// TwinCAT 3 PLC project HFM
// ProgramVersion: 3.1.4024.0
// libraries:
//   Tc2_Standard, * (Beckhoff Automation GmbH)
//   Tc2_System, * (Beckhoff Automation GmbH)
//   Tc3_Module, * (Beckhoff Automation GmbH)
//   LCLS General,0.0.0,SLAC
//   lcls-twincat-motion,0.0.0,SLAC
//   PMPS,0.0.0,SLAC - LCLS
//   TcUnit,1.3.0.0,www.tcunit.org
// project tree:
//   / PlcTask.TcTTO
//   POUs/ MAIN.TcPOU
// real-time tasks:
//   TASK PlcTask: cycle T#10ms, priority 20, ADS port 350
// motion (NC):
//   TASK NC-Task 1 SAF: cycle T#2ms, priority 4, ADS port 501
//   TASK NC-Task 1 SVB: cycle T#10ms, priority 8, ADS port 511
//   AXIS Axis 1(HFM-Y1) (id 1)
//     Dynamic: AccelerationMaximum=20, DecelerationMaximum=20, Acceleration=0.742063, Deceleration=0.742063, Jerk=275.329
//     Velo: RefSearch=5, RefSync=5, SlowManual=5, FastManual=5, Maximum=0.2
//     PositionAreaControl: Range=0.0002
//     MotionControl: Range=0.5, Time=1
//     TargetPosControl: Range=0.0001
//     PEHControl: Time=0.1
//     OtherSettings: AllowMotionCmdToSlave=true, PulseDistancePos=0.5, PulseDistanceNeg=0.5
//     encoder EncType=4
//       EncPara: ScaleFactorNumerator=0.0002, Inverse=true, MaxCount=#xffffffff
//     drive DrvType=5
//       DrvPara: Inverse=true
//         Analog: VeloReferenz=20, TorqueSetpointScale=10, ScaleFactorActTorque=0.1
//         TimeComp: TaskDelayCycles=1
//     controller CtrType=1
//       CtrPara: PriorControlFactor=1
//         PosDiffControl: Range=1
//         PID: PosKp=22
//         Observer: BandWidth=20
//   AXIS Axis 2(HFM-Y2) (id 2)
//     Dynamic: AccelerationMaximum=20, DecelerationMaximum=20, Acceleration=0.75757, Deceleration=0.75757, Jerk=286.956
//     Velo: RefSearch=5, RefSync=5, SlowManual=5, FastManual=5, Maximum=0.2
//     PositionAreaControl: Range=0.0002
//     TargetPosControl: Range=0.0001
//     OtherSettings: AllowMotionCmdToSlave=true, PulseDistancePos=0.5, PulseDistanceNeg=0.5
//     encoder EncType=4
//       EncPara: ScaleFactorNumerator=0.0002, Inverse=true, MaxCount=#xffffffff
//     drive DrvType=5
//       DrvPara: Inverse=true
//         Analog: VeloReferenz=20, TorqueSetpointScale=10, ScaleFactorActTorque=0.1
//         TimeComp: TaskDelayCycles=1
//     controller CtrType=1
//       CtrPara: PriorControlFactor=1
//         PosDiffControl: Range=2
//         PID: PosKp=22
//         Observer: BandWidth=20
//   AXIS Axis 3(HFM-Y3) (id 3)
//     Dynamic: AccelerationMaximum=20, DecelerationMaximum=20, Acceleration=0.742063, Deceleration=0.742063, Jerk=275.329
//     Velo: RefSearch=5, RefSync=5, SlowManual=5, FastManual=5, Maximum=0.2
//     PositionAreaControl: Range=0.0002
//     TargetPosControl: Range=0.0001
//     OtherSettings: AllowMotionCmdToSlave=true, PulseDistancePos=0.5, PulseDistanceNeg=0.5
//     encoder EncType=4
//       EncPara: ScaleFactorNumerator=0.0002, Inverse=true, MaxCount=#xffffffff
//     drive DrvType=5
//       DrvPara: Inverse=true
//         Analog: VeloReferenz=20, TorqueSetpointScale=10, ScaleFactorActTorque=0.1
//         TimeComp: TaskDelayCycles=1
//     controller CtrType=1
//       CtrPara: PriorControlFactor=1
//         PosDiffControl: Range=2
//         PID: PosKp=22
//         Observer: BandWidth=20
//   AXIS Axis 4(HFM-X1) (id 4)
//     Dynamic: AccelerationMaximum=20, DecelerationMaximum=20, Acceleration=6.71181, Deceleration=6.71181, Jerk=22524.2
//     Velo: RefSearch=5, RefSync=5, SlowManual=5, FastManual=5, Maximum=0.2
//     PositionAreaControl: Range=2e-05
//     TargetPosControl: Range=1e-05
//     OtherSettings: AllowMotionCmdToSlave=true, PulseDistancePos=0.5, PulseDistanceNeg=0.5
//     encoder EncType=4
//       EncPara: ScaleFactorNumerator=2e-05, MaxCount=#xffffffff
//     drive DrvType=5
//       Analog: VeloReferenz=20, TorqueSetpointScale=10, ScaleFactorActTorque=0.1
//       TimeComp: TaskDelayCycles=1
//     controller CtrType=1
//       CtrPara: PriorControlFactor=1
//         PID: PosKp=50
//         Observer: BandWidth=20
//   AXIS Axis 5(HFM-X2) (id 5)
//     Dynamic: AccelerationMaximum=20, DecelerationMaximum=20, Acceleration=3.45558, Deceleration=3.45558, Jerk=5970.51
//     Velo: RefSearch=5, RefSync=5, SlowManual=5, FastManual=5, Maximum=0.2
//     PositionAreaControl: Range=2e-05
//     TargetPosControl: Range=1e-05
//     OtherSettings: AllowMotionCmdToSlave=true, PulseDistancePos=0.5, PulseDistanceNeg=0.5
//     encoder EncType=4
//       EncPara: ScaleFactorNumerator=2e-05, MaxCount=#xffffffff
//     drive DrvType=5
//       Analog: VeloReferenz=20, TorqueSetpointScale=10, ScaleFactorActTorque=0.1
//       TimeComp: TaskDelayCycles=1
//     controller CtrType=1
//       CtrPara: PriorControlFactor=1
//         PID: PosKp=50
//         Observer: BandWidth=20
//   AXIS Axis 6(FM-Y1) (id 6)
//     Dynamic: AccelerationMaximum=20, DecelerationMaximum=20, Acceleration=0.742063, Deceleration=0.742063, Jerk=275.329
//     Velo: RefSearch=1, RefSync=1, SlowManual=1, FastManual=1, Maximum=0.2
//     PositionAreaControl: Range=0.0002
//     TargetPosControl: Range=0.0001
//     OtherSettings: AllowMotionCmdToSlave=true, PulseDistancePos=0.5, PulseDistanceNeg=0.5
//     encoder EncType=4
//       EncPara: ScaleFactorNumerator=0.0002, Inverse=true, MaxCount=#xffffffff
//     drive DrvType=5
//       DrvPara: Inverse=true
//         Analog: VeloReferenz=20, TorqueSetpointScale=10, ScaleFactorActTorque=0.1
//         TimeComp: TaskDelayCycles=1
//     controller CtrType=1
//       CtrPara: PriorControlFactor=1
//         PosDiffControl: Range=1
//         PID: PosKp=22
//         Observer: BandWidth=20
//   AXIS Axis 7(FM-Y2) (id 7)
//     Dynamic: AccelerationMaximum=20, DecelerationMaximum=20, Acceleration=0.742063, Deceleration=0.742063, Jerk=275.329
//     Velo: RefSearch=1, RefSync=1, SlowManual=1, FastManual=1, Maximum=0.2
//     PositionAreaControl: Range=0.0002
//     TargetPosControl: Range=0.0001
//     OtherSettings: AllowMotionCmdToSlave=true, PulseDistancePos=0.5, PulseDistanceNeg=0.5
//     encoder EncType=4
//       EncPara: ScaleFactorNumerator=0.0002, Inverse=true, MaxCount=#xffffffff
//     drive DrvType=5
//       DrvPara: Inverse=true
//         Analog: VeloReferenz=20, TorqueSetpointScale=10, ScaleFactorActTorque=0.1
//         TimeComp: TaskDelayCycles=1
//     controller CtrType=1
//       CtrPara: PriorControlFactor=1
//         PosDiffControl: Range=1
//         PID: PosKp=22
//         Observer: BandWidth=20
//   AXIS Axis 8(FM-Y3) (id 8)
//     Dynamic: AccelerationMaximum=20, DecelerationMaximum=20, Acceleration=0.742063, Deceleration=0.742063, Jerk=275.329
//     Velo: RefSearch=1, RefSync=1, SlowManual=1, FastManual=1, Maximum=0.2
//     PositionAreaControl: Range=0.0002
//     TargetPosControl: Range=0.0001
//     OtherSettings: AllowMotionCmdToSlave=true, PulseDistancePos=0.5, PulseDistanceNeg=0.5
//     encoder EncType=4
//       EncPara: ScaleFactorNumerator=0.0002, Inverse=true, MaxCount=#xffffffff
//     drive DrvType=5
//       DrvPara: Inverse=true
//         Analog: VeloReferenz=20, TorqueSetpointScale=10, ScaleFactorActTorque=0.1
//         TimeComp: TaskDelayCycles=1
//     controller CtrType=1
//       CtrPara: PriorControlFactor=1
//         PosDiffControl: Range=1
//         PID: PosKp=22
//         Observer: BandWidth=20
//   AXIS Axis 9(FM-X1) (id 9)
//     Dynamic: AccelerationMaximum=20, DecelerationMaximum=20, Acceleration=6.71181, Deceleration=6.71181, Jerk=22524.2
//     Velo: RefSearch=1, RefSync=1, SlowManual=1, FastManual=1, Maximum=0.2
//     PositionAreaControl: Range=2e-05
//     TargetPosControl: Range=1e-05
//     OtherSettings: AllowMotionCmdToSlave=true, PulseDistancePos=0.5, PulseDistanceNeg=0.5
//     encoder EncType=4
//       EncPara: ScaleFactorNumerator=2e-05, MaxCount=#xffffffff
//     drive DrvType=5
//       Analog: VeloReferenz=20, TorqueSetpointScale=10, ScaleFactorActTorque=0.1
//       TimeComp: TaskDelayCycles=1
//     controller CtrType=1
//       CtrPara: PriorControlFactor=1
//         PID: PosKp=50
//         Observer: BandWidth=20
//   AXIS Axis 10(FM-X2) (id 10)
//     Dynamic: AccelerationMaximum=20, DecelerationMaximum=20, Acceleration=6.71181, Deceleration=6.71181, Jerk=22524.2
//     Velo: RefSearch=1, RefSync=1, SlowManual=1, FastManual=1, Maximum=0.2
//     PositionAreaControl: Range=2e-05
//     TargetPosControl: Range=1e-05
//     OtherSettings: AllowMotionCmdToSlave=true, PulseDistancePos=0.5, PulseDistanceNeg=0.5
//     encoder EncType=4
//       EncPara: ScaleFactorNumerator=2e-05, MaxCount=#xffffffff
//     drive DrvType=5
//       Analog: VeloReferenz=20, TorqueSetpointScale=10, ScaleFactorActTorque=0.1
//       TimeComp: TaskDelayCycles=1
//     controller CtrType=1
//       CtrPara: PriorControlFactor=1
//         PID: PosKp=50
//         Observer: BandWidth=20
// I/O:
//   DEVICE Device 3 (EtherCAT), AmsNetId 169.254.61.1.4.1
//     Term 1 (EK1100) [EK1100 EtherCAT Coupler (2A E-Bus)]
//       Term 2 (EL2522) [EL2522 2Ch. Pulse Train Output]
//       Term 3 (EL5112) [EL5112 2Ch. Inc. Encoder 5V (2xAB or 1xABC RS422,TTL)]
//       Term 4 (EL2522) [EL2522 2Ch. Pulse Train Output]
//       Term 5 (EL5112) [EL5112 2Ch. Inc. Encoder 5V (2xAB or 1xABC RS422,TTL)]
//       Term 6 (EL2522) [EL2522 2Ch. Pulse Train Output]
//       Term 7 (EL1889) [EL1889 16Ch. Dig. Input 24V, 3ms, negative]
//       Term 8 (EL9011) [EL9011 End Terminal]
//   DEVICE Device 1 (EtherCAT), AmsNetId 192.168.61.50.2.1
//     Term 9 (EK1100) [EK1100 EtherCAT Coupler (2A E-Bus)]
//       Term 10 (EL2522) [EL2522 2Ch. Pulse Train Output]
//       Term 11 (EL5112) [EL5112 2Ch. Inc. Encoder 5V (2xAB or 1xABC RS422,TTL)]
//       Term 12 (EL2522) [EL2522 2Ch. Pulse Train Output]
//       Term 13 (EL5112) [EL5112 2Ch. Inc. Encoder 5V (2xAB or 1xABC RS422,TTL)]
//       Term 14 (EL2522) [EL2522 2Ch. Pulse Train Output]
//       Term 15 (EL1889) [EL1889 16Ch. Dig. Input 24V, 3ms, negative]
//       Term 8 (EL9011) [EL9011 End Terminal]
// variable links:
//   NC-Task 1 SAF/Axes/Axis 10(FM-X2) <-> Device 1 (EtherCAT)/Term 9 (EK1100)/Term 14 (EL2522)
//     Drive/Inputs/In/nState1 @bit 6 <-> PTO Status Channel 1/Status/Error
//     Drive/Inputs/In/nState1 @bit 1 <-> PTO Status Channel 1/Status/Ramp active
//     Drive/Inputs/In/nState1 <-> PTO Status Channel 1/Status/Sel. Ack/End counter
//     Drive/Inputs/In/nState2 @bit 5 <-> PTO Status Channel 1/Status/Sync error
//     Drive/Inputs/In/nState2 @bit 7 <-> PTO Status Channel 1/Status/TxPDO Toggle
//     Drive/Inputs/In/nState4 @bit 1 <-> WcState/InputToggle
//     Drive/Inputs/In/nState4 <-> WcState/WcState
//     Drive/Outputs/Out/nCtrl1 @bit 1 <-> PTO Control Channel 1/Control/Disable ramp
//     Drive/Outputs/Out/nCtrl1 <-> PTO Control Channel 1/Control/Frequency select
//     Drive/Outputs/Out/nCtrl1 @bit 2 <-> PTO Control Channel 1/Control/Go counter
//     Drive/Outputs/Out/nDataOut1[0] <-> PTO Control Channel 1/Frequency value
//     Drive/Outputs/Out/nDataOut5 <-> PTO Target Channel 1/Target counter value
//     Enc/Inputs/In/nDataIn1 <-> ENC Status Channel 1/Counter value
//     Enc/Inputs/In/nState1 @bit 4 <-> ENC Status Channel 1/Status/Counter overflow
//     Enc/Inputs/In/nState1 @bit 3 <-> ENC Status Channel 1/Status/Counter underflow
//     Enc/Inputs/In/nState1 @bit 2 <-> ENC Status Channel 1/Status/Set counter done
//     Enc/Inputs/In/nState2 @bit 5 <-> ENC Status Channel 1/Status/Sync error
//     Enc/Inputs/In/nState2 @bit 6 <-> ENC Status Channel 1/Status/TxPDO State
//     Enc/Inputs/In/nState2 @bit 7 <-> ENC Status Channel 1/Status/TxPDO Toggle
//     Enc/Inputs/In/nState4 @bit 1 <-> WcState/InputToggle
//     Enc/Inputs/In/nState4 <-> WcState/WcState
//     Enc/Outputs/Out/nCtrl1 @bit 2 <-> ENC Control Channel 1/Control/Set counter
//     Enc/Outputs/Out/nCtrl2 @bit 7 <-> ENC Control Channel 1/Control/Reserved
//     Enc/Outputs/Out/nDataOut1 <-> ENC Control Channel 1/Set counter value
//   NC-Task 1 SAF/Axes/Axis 2(HFM-Y2) <-> Device 3 (EtherCAT)/Term 1 (EK1100)/Term 2 (EL2522)
//     Drive/Inputs/In/nState1 @bit 6 <-> PTO Status Channel 2/Status/Error
//     Drive/Inputs/In/nState1 @bit 1 <-> PTO Status Channel 2/Status/Ramp active
//     Drive/Inputs/In/nState1 <-> PTO Status Channel 2/Status/Sel. Ack/End counter
//     Drive/Inputs/In/nState2 @bit 5 <-> PTO Status Channel 2/Status/Sync error
//     Drive/Inputs/In/nState2 @bit 7 <-> PTO Status Channel 2/Status/TxPDO Toggle
//     Drive/Inputs/In/nState4 @bit 1 <-> WcState/InputToggle
//     Drive/Inputs/In/nState4 <-> WcState/WcState
//     Drive/Outputs/Out/nCtrl1 @bit 1 <-> PTO Control Channel 2/Control/Disable ramp
//     Drive/Outputs/Out/nCtrl1 <-> PTO Control Channel 2/Control/Frequency select
//     Drive/Outputs/Out/nCtrl1 @bit 2 <-> PTO Control Channel 2/Control/Go counter
//     Drive/Outputs/Out/nDataOut1[0] <-> PTO Control Channel 2/Frequency value
//     Drive/Outputs/Out/nDataOut5 <-> PTO Target Channel 2/Target counter value
//   NC-Task 1 SAF/Axes/Axis 2(HFM-Y2) <-> Device 3 (EtherCAT)/Term 1 (EK1100)/Term 3 (EL5112)
//     Enc/Inputs/In/nDataIn1 <-> ENC Status Channel 2/Counter value
//     Enc/Inputs/In/nDataIn2 <-> ENC Status Channel 2/Latch value
//     Enc/Inputs/In/nState1 @bit 4 <-> ENC Status Channel 2/Status/Counter overflow
//     Enc/Inputs/In/nState1 @bit 3 <-> ENC Status Channel 2/Status/Counter underflow
//     Enc/Inputs/In/nState1 @bit 1 <-> ENC Status Channel 2/Status/Latch extern valid
//     Enc/Inputs/In/nState1 @bit 6 <-> ENC Status Channel 2/Status/Open circuit
//     Enc/Inputs/In/nState1 @bit 2 <-> ENC Status Channel 2/Status/Set counter done
//     Enc/Inputs/In/nState2 @bit 4 <-> ENC Status Channel 2/Status/Diag
//     Enc/Inputs/In/nState2 @bit 6 <-> ENC Status Channel 2/Status/Input cycle counter
//     Enc/Inputs/In/nState2 <-> ENC Status Channel 2/Status/Status of input A
//     Enc/Inputs/In/nState2 @bit 1 <-> ENC Status Channel 2/Status/Status of input B
//     Enc/Inputs/In/nState2 @bit 3 <-> ENC Status Channel 2/Status/Status of input gate
//     Enc/Inputs/In/nState2 @bit 5 <-> ENC Status Channel 2/Status/TxPDO State
//     Enc/Inputs/In/nState3 @bit 4 <-> ENC Status Channel 2/Status/Counter value out of range
//     Enc/Inputs/In/nState3 <-> ENC Status Channel 2/Status/Software gate valid
//     Enc/Inputs/In/nState4 @bit 1 <-> WcState/InputToggle
//     Enc/Inputs/In/nState4 <-> WcState/WcState
//     Enc/Outputs/Out/nCtrl1 @bit 3 <-> ENC Control Channel 2/Control/Enable latch extern on negative edge
//     Enc/Outputs/Out/nCtrl1 @bit 1 <-> ENC Control Channel 2/Control/Enable latch extern on positive edge
//     Enc/Outputs/Out/nCtrl1 @bit 2 <-> ENC Control Channel 2/Control/Set counter
//     Enc/Outputs/Out/nCtrl2 @bit 2 <-> ENC Control Channel 2/Control/Set counter on latch extern on negative edge
//     Enc/Outputs/Out/nCtrl2 @bit 1 <-> ENC Control Channel 2/Control/Set counter on latch extern on positive edge
//     Enc/Outputs/Out/nCtrl2 <-> ENC Control Channel 2/Control/Set software gate
//     Enc/Outputs/Out/nDataOut1 <-> ENC Control Channel 2/Set counter value
//   NC-Task 1 SAF/Axes/Axis 3(HFM-Y3) <-> Device 3 (EtherCAT)/Term 1 (EK1100)/Term 4 (EL2522)
//     Drive/Inputs/In/nState1 @bit 6 <-> PTO Status Channel 1/Status/Error
//     Drive/Inputs/In/nState1 @bit 1 <-> PTO Status Channel 1/Status/Ramp active
//     Drive/Inputs/In/nState1 <-> PTO Status Channel 1/Status/Sel. Ack/End counter
//     Drive/Inputs/In/nState2 @bit 5 <-> PTO Status Channel 1/Status/Sync error
//     Drive/Inputs/In/nState2 @bit 7 <-> PTO Status Channel 1/Status/TxPDO Toggle
//     Drive/Inputs/In/nState4 @bit 1 <-> WcState/InputToggle
//     Drive/Inputs/In/nState4 <-> WcState/WcState
//     Drive/Outputs/Out/nCtrl1 @bit 1 <-> PTO Control Channel 1/Control/Disable ramp
//     Drive/Outputs/Out/nCtrl1 <-> PTO Control Channel 1/Control/Frequency select
//     Drive/Outputs/Out/nCtrl1 @bit 2 <-> PTO Control Channel 1/Control/Go counter
//     Drive/Outputs/Out/nDataOut1[0] <-> PTO Control Channel 1/Frequency value
//     Drive/Outputs/Out/nDataOut5 <-> PTO Target Channel 1/Target counter value
//   NC-Task 1 SAF/Axes/Axis 3(HFM-Y3) <-> Device 3 (EtherCAT)/Term 1 (EK1100)/Term 5 (EL5112)
//     Enc/Inputs/In/nDataIn1 <-> ENC Status Channel 1/Counter value
//     Enc/Inputs/In/nDataIn2 <-> ENC Status Channel 1/Latch value
//     Enc/Inputs/In/nState1 @bit 4 <-> ENC Status Channel 1/Status/Counter overflow
//     Enc/Inputs/In/nState1 @bit 3 <-> ENC Status Channel 1/Status/Counter underflow
//     Enc/Inputs/In/nState1 @bit 7 <-> ENC Status Channel 1/Status/Extrapolation stall
//     Enc/Inputs/In/nState1 <-> ENC Status Channel 1/Status/Latch C valid
//     Enc/Inputs/In/nState1 @bit 1 <-> ENC Status Channel 1/Status/Latch extern valid
//     Enc/Inputs/In/nState1 @bit 6 <-> ENC Status Channel 1/Status/Open circuit
//     Enc/Inputs/In/nState1 @bit 2 <-> ENC Status Channel 1/Status/Set counter done
//     Enc/Inputs/In/nState1 @bit 5 <-> ENC Status Channel 1/Status/Status of input status
//     Enc/Inputs/In/nState2 @bit 4 <-> ENC Status Channel 1/Status/Diag
//     Enc/Inputs/In/nState2 @bit 6 <-> ENC Status Channel 1/Status/Input cycle counter
//     Enc/Inputs/In/nState2 <-> ENC Status Channel 1/Status/Status of input A
//     Enc/Inputs/In/nState2 @bit 1 <-> ENC Status Channel 1/Status/Status of input B
//     Enc/Inputs/In/nState2 @bit 2 <-> ENC Status Channel 1/Status/Status of input C
//     Enc/Inputs/In/nState2 @bit 3 <-> ENC Status Channel 1/Status/Status of input gate
//     Enc/Inputs/In/nState2 @bit 5 <-> ENC Status Channel 1/Status/TxPDO State
//     Enc/Inputs/In/nState3 @bit 4 <-> ENC Status Channel 1/Status/Counter value out of range
//     Enc/Inputs/In/nState3 @bit 2 <-> ENC Status Channel 1/Status/Direction inversion detected
//     Enc/Inputs/In/nState3 @bit 1 <-> ENC Status Channel 1/Status/Latch extern 2 valid
//     Enc/Inputs/In/nState3 <-> ENC Status Channel 1/Status/Software gate valid
//     Enc/Inputs/In/nState3 @bit 3 <-> ENC Status Channel 1/Status/Status of extern latch
//     Enc/Inputs/In/nState4 @bit 1 <-> WcState/InputToggle
//     Enc/Inputs/In/nState4 <-> WcState/WcState
//     Enc/Outputs/Out/nCtrl1 <-> ENC Control Channel 1/Control/Enable latch C
//     Enc/Outputs/Out/nCtrl1 @bit 3 <-> ENC Control Channel 1/Control/Enable latch extern on negative edge
//     Enc/Outputs/Out/nCtrl1 @bit 1 <-> ENC Control Channel 1/Control/Enable latch extern on positive edge
//     Enc/Outputs/Out/nCtrl1 @bit 2 <-> ENC Control Channel 1/Control/Set counter
//     Enc/Outputs/Out/nCtrl1 @bit 7 <-> ENC Control Channel 1/Control/Set counter on latch C
//     Enc/Outputs/Out/nCtrl2 @bit 4 <-> ENC Control Channel 1/Control/Enable latch extern 2 on negative edge
//     Enc/Outputs/Out/nCtrl2 @bit 3 <-> ENC Control Channel 1/Control/Enable latch extern 2 on positive edge
//     Enc/Outputs/Out/nCtrl2 @bit 2 <-> ENC Control Channel 1/Control/Set counter on latch extern on negative edge
//     Enc/Outputs/Out/nCtrl2 @bit 1 <-> ENC Control Channel 1/Control/Set counter on latch extern on positive edge
//     Enc/Outputs/Out/nCtrl2 <-> ENC Control Channel 1/Control/Set software gate
//     Enc/Outputs/Out/nDataOut1 <-> ENC Control Channel 1/Set counter value
//   NC-Task 1 SAF/Axes/Axis 4(HFM-X1) <-> Device 3 (EtherCAT)/Term 1 (EK1100)/Term 4 (EL2522)
//     Drive/Inputs/In/nState1 @bit 6 <-> PTO Status Channel 2/Status/Error
//     Drive/Inputs/In/nState1 @bit 1 <-> PTO Status Channel 2/Status/Ramp active
//     Drive/Inputs/In/nState1 <-> PTO Status Channel 2/Status/Sel. Ack/End counter
//     Drive/Inputs/In/nState2 @bit 5 <-> PTO Status Channel 2/Status/Sync error
//     Drive/Inputs/In/nState2 @bit 7 <-> PTO Status Channel 2/Status/TxPDO Toggle
//     Drive/Inputs/In/nState4 @bit 1 <-> WcState/InputToggle
//     Drive/Inputs/In/nState4 <-> WcState/WcState
//     Drive/Outputs/Out/nCtrl1 @bit 1 <-> PTO Control Channel 2/Control/Disable ramp
//     Drive/Outputs/Out/nCtrl1 <-> PTO Control Channel 2/Control/Frequency select
//     Drive/Outputs/Out/nCtrl1 @bit 2 <-> PTO Control Channel 2/Control/Go counter
//     Drive/Outputs/Out/nDataOut1[0] <-> PTO Control Channel 2/Frequency value
//     Drive/Outputs/Out/nDataOut5 <-> PTO Target Channel 2/Target counter value
//     Enc/Inputs/In/nDataIn1 <-> ENC Status Channel 2/Counter value
//     Enc/Inputs/In/nState1 @bit 4 <-> ENC Status Channel 2/Status/Counter overflow
//     Enc/Inputs/In/nState1 @bit 3 <-> ENC Status Channel 2/Status/Counter underflow
//     Enc/Inputs/In/nState1 @bit 2 <-> ENC Status Channel 2/Status/Set counter done
//     Enc/Inputs/In/nState2 @bit 5 <-> ENC Status Channel 2/Status/Sync error
//     Enc/Inputs/In/nState2 @bit 6 <-> ENC Status Channel 2/Status/TxPDO State
//     Enc/Inputs/In/nState2 @bit 7 <-> ENC Status Channel 2/Status/TxPDO Toggle
//     Enc/Inputs/In/nState4 @bit 1 <-> WcState/InputToggle
//     Enc/Inputs/In/nState4 <-> WcState/WcState
//     Enc/Outputs/Out/nCtrl1 @bit 2 <-> ENC Control Channel 2/Control/Set counter
//     Enc/Outputs/Out/nCtrl2 @bit 7 <-> ENC Control Channel 2/Control/Reserved
//     Enc/Outputs/Out/nDataOut1 <-> ENC Control Channel 2/Set counter value
//   NC-Task 1 SAF/Axes/Axis 5(HFM-X2) <-> Device 3 (EtherCAT)/Term 1 (EK1100)/Term 6 (EL2522)
//     Drive/Inputs/In/nState1 @bit 6 <-> PTO Status Channel 1/Status/Error
//     Drive/Inputs/In/nState1 @bit 1 <-> PTO Status Channel 1/Status/Ramp active
//     Drive/Inputs/In/nState1 <-> PTO Status Channel 1/Status/Sel. Ack/End counter
//     Drive/Inputs/In/nState2 @bit 5 <-> PTO Status Channel 1/Status/Sync error
//     Drive/Inputs/In/nState2 @bit 7 <-> PTO Status Channel 1/Status/TxPDO Toggle
//     Drive/Inputs/In/nState4 @bit 1 <-> WcState/InputToggle
//     Drive/Inputs/In/nState4 <-> WcState/WcState
//     Drive/Outputs/Out/nCtrl1 @bit 1 <-> PTO Control Channel 1/Control/Disable ramp
//     Drive/Outputs/Out/nCtrl1 <-> PTO Control Channel 1/Control/Frequency select
//     Drive/Outputs/Out/nCtrl1 @bit 2 <-> PTO Control Channel 1/Control/Go counter
//     Drive/Outputs/Out/nDataOut1[0] <-> PTO Control Channel 1/Frequency value
//     Drive/Outputs/Out/nDataOut5 <-> PTO Target Channel 1/Target counter value
//     Enc/Inputs/In/nDataIn1 <-> ENC Status Channel 1/Counter value
//     Enc/Inputs/In/nState1 @bit 4 <-> ENC Status Channel 1/Status/Counter overflow
//     Enc/Inputs/In/nState1 @bit 3 <-> ENC Status Channel 1/Status/Counter underflow
//     Enc/Inputs/In/nState1 @bit 2 <-> ENC Status Channel 1/Status/Set counter done
//     Enc/Inputs/In/nState2 @bit 5 <-> ENC Status Channel 1/Status/Sync error
//     Enc/Inputs/In/nState2 @bit 6 <-> ENC Status Channel 1/Status/TxPDO State
//     Enc/Inputs/In/nState2 @bit 7 <-> ENC Status Channel 1/Status/TxPDO Toggle
//     Enc/Inputs/In/nState4 @bit 1 <-> WcState/InputToggle
//     Enc/Inputs/In/nState4 <-> WcState/WcState
//     Enc/Outputs/Out/nCtrl1 @bit 2 <-> ENC Control Channel 1/Control/Set counter
//     Enc/Outputs/Out/nCtrl2 @bit 7 <-> ENC Control Channel 1/Control/Reserved
//     Enc/Outputs/Out/nDataOut1 <-> ENC Control Channel 1/Set counter value
//   NC-Task 1 SAF/Axes/Axis 6(FM-Y1) <-> Device 1 (EtherCAT)/Term 9 (EK1100)/Term 10 (EL2522)
//     Drive/Inputs/In/nState1 @bit 6 <-> PTO Status Channel 1/Status/Error
//     Drive/Inputs/In/nState1 @bit 1 <-> PTO Status Channel 1/Status/Ramp active
//     Drive/Inputs/In/nState1 <-> PTO Status Channel 1/Status/Sel. Ack/End counter
//     Drive/Inputs/In/nState2 @bit 5 <-> PTO Status Channel 1/Status/Sync error
//     Drive/Inputs/In/nState2 @bit 7 <-> PTO Status Channel 1/Status/TxPDO Toggle
//     Drive/Inputs/In/nState4 @bit 1 <-> WcState/InputToggle
//     Drive/Inputs/In/nState4 <-> WcState/WcState
//     Drive/Outputs/Out/nCtrl1 @bit 1 <-> PTO Control Channel 1/Control/Disable ramp
//     Drive/Outputs/Out/nCtrl1 <-> PTO Control Channel 1/Control/Frequency select
//     Drive/Outputs/Out/nCtrl1 @bit 2 <-> PTO Control Channel 1/Control/Go counter
//     Drive/Outputs/Out/nDataOut1[0] <-> PTO Control Channel 1/Frequency value
//     Drive/Outputs/Out/nDataOut5 <-> PTO Target Channel 1/Target counter value
//   NC-Task 1 SAF/Axes/Axis 6(FM-Y1) <-> Device 1 (EtherCAT)/Term 9 (EK1100)/Term 11 (EL5112)
//     Enc/Inputs/In/nDataIn1 <-> ENC Status Channel 1/Counter value
//     Enc/Inputs/In/nDataIn2 <-> ENC Status Channel 1/Latch value
//     Enc/Inputs/In/nState1 @bit 4 <-> ENC Status Channel 1/Status/Counter overflow
//     Enc/Inputs/In/nState1 @bit 3 <-> ENC Status Channel 1/Status/Counter underflow
//     Enc/Inputs/In/nState1 @bit 1 <-> ENC Status Channel 1/Status/Latch extern valid
//     Enc/Inputs/In/nState1 @bit 6 <-> ENC Status Channel 1/Status/Open circuit
//     Enc/Inputs/In/nState1 @bit 2 <-> ENC Status Channel 1/Status/Set counter done
//     Enc/Inputs/In/nState2 @bit 4 <-> ENC Status Channel 1/Status/Diag
//     Enc/Inputs/In/nState2 @bit 6 <-> ENC Status Channel 1/Status/Input cycle counter
//     Enc/Inputs/In/nState2 <-> ENC Status Channel 1/Status/Status of input A
//     Enc/Inputs/In/nState2 @bit 1 <-> ENC Status Channel 1/Status/Status of input B
//     Enc/Inputs/In/nState2 @bit 3 <-> ENC Status Channel 1/Status/Status of input gate
//     Enc/Inputs/In/nState2 @bit 5 <-> ENC Status Channel 1/Status/TxPDO State
//     Enc/Inputs/In/nState3 @bit 4 <-> ENC Status Channel 1/Status/Counter value out of range
//     Enc/Inputs/In/nState3 <-> ENC Status Channel 1/Status/Software gate valid
//     Enc/Inputs/In/nState4 @bit 1 <-> WcState/InputToggle
//     Enc/Inputs/In/nState4 <-> WcState/WcState
//     Enc/Outputs/Out/nCtrl1 @bit 3 <-> ENC Control Channel 1/Control/Enable latch extern on negative edge
//     Enc/Outputs/Out/nCtrl1 @bit 1 <-> ENC Control Channel 1/Control/Enable latch extern on positive edge
//     Enc/Outputs/Out/nCtrl1 @bit 2 <-> ENC Control Channel 1/Control/Set counter
//     Enc/Outputs/Out/nCtrl2 @bit 2 <-> ENC Control Channel 1/Control/Set counter on latch extern on negative edge
//     Enc/Outputs/Out/nCtrl2 @bit 1 <-> ENC Control Channel 1/Control/Set counter on latch extern on positive edge
//     Enc/Outputs/Out/nCtrl2 <-> ENC Control Channel 1/Control/Set software gate
//     Enc/Outputs/Out/nDataOut1 <-> ENC Control Channel 1/Set counter value
//   NC-Task 1 SAF/Axes/Axis 7(FM-Y2) <-> Device 1 (EtherCAT)/Term 9 (EK1100)/Term 10 (EL2522)
//     Drive/Inputs/In/nState1 @bit 6 <-> PTO Status Channel 2/Status/Error
//     Drive/Inputs/In/nState1 @bit 1 <-> PTO Status Channel 2/Status/Ramp active
//     Drive/Inputs/In/nState1 <-> PTO Status Channel 2/Status/Sel. Ack/End counter
//     Drive/Inputs/In/nState2 @bit 5 <-> PTO Status Channel 2/Status/Sync error
//     Drive/Inputs/In/nState2 @bit 7 <-> PTO Status Channel 2/Status/TxPDO Toggle
//     Drive/Inputs/In/nState4 @bit 1 <-> WcState/InputToggle
//     Drive/Inputs/In/nState4 <-> WcState/WcState
//     Drive/Outputs/Out/nCtrl1 @bit 1 <-> PTO Control Channel 2/Control/Disable ramp
//     Drive/Outputs/Out/nCtrl1 <-> PTO Control Channel 2/Control/Frequency select
//     Drive/Outputs/Out/nCtrl1 @bit 2 <-> PTO Control Channel 2/Control/Go counter
//     Drive/Outputs/Out/nDataOut1[0] <-> PTO Control Channel 2/Frequency value
//     Drive/Outputs/Out/nDataOut5 <-> PTO Target Channel 2/Target counter value
//   NC-Task 1 SAF/Axes/Axis 7(FM-Y2) <-> Device 1 (EtherCAT)/Term 9 (EK1100)/Term 11 (EL5112)
//     Enc/Inputs/In/nDataIn1 <-> ENC Status Channel 2/Counter value
//     Enc/Inputs/In/nDataIn2 <-> ENC Status Channel 2/Latch value
//     Enc/Inputs/In/nState1 @bit 4 <-> ENC Status Channel 2/Status/Counter overflow
//     Enc/Inputs/In/nState1 @bit 3 <-> ENC Status Channel 2/Status/Counter underflow
//     Enc/Inputs/In/nState1 @bit 1 <-> ENC Status Channel 2/Status/Latch extern valid
//     Enc/Inputs/In/nState1 @bit 6 <-> ENC Status Channel 2/Status/Open circuit
//     Enc/Inputs/In/nState1 @bit 2 <-> ENC Status Channel 2/Status/Set counter done
//     Enc/Inputs/In/nState2 @bit 4 <-> ENC Status Channel 2/Status/Diag
//     Enc/Inputs/In/nState2 @bit 6 <-> ENC Status Channel 2/Status/Input cycle counter
//     Enc/Inputs/In/nState2 <-> ENC Status Channel 2/Status/Status of input A
//     Enc/Inputs/In/nState2 @bit 1 <-> ENC Status Channel 2/Status/Status of input B
//     Enc/Inputs/In/nState2 @bit 3 <-> ENC Status Channel 2/Status/Status of input gate
//     Enc/Inputs/In/nState2 @bit 5 <-> ENC Status Channel 2/Status/TxPDO State
//     Enc/Inputs/In/nState3 @bit 4 <-> ENC Status Channel 2/Status/Counter value out of range
//     Enc/Inputs/In/nState3 <-> ENC Status Channel 2/Status/Software gate valid
//     Enc/Inputs/In/nState4 @bit 1 <-> WcState/InputToggle
//     Enc/Inputs/In/nState4 <-> WcState/WcState
//     Enc/Outputs/Out/nCtrl1 @bit 3 <-> ENC Control Channel 2/Control/Enable latch extern on negative edge
//     Enc/Outputs/Out/nCtrl1 @bit 1 <-> ENC Control Channel 2/Control/Enable latch extern on positive edge
//     Enc/Outputs/Out/nCtrl1 @bit 2 <-> ENC Control Channel 2/Control/Set counter
//     Enc/Outputs/Out/nCtrl2 @bit 2 <-> ENC Control Channel 2/Control/Set counter on latch extern on negative edge
//     Enc/Outputs/Out/nCtrl2 @bit 1 <-> ENC Control Channel 2/Control/Set counter on latch extern on positive edge
//     Enc/Outputs/Out/nCtrl2 <-> ENC Control Channel 2/Control/Set software gate
//     Enc/Outputs/Out/nDataOut1 <-> ENC Control Channel 2/Set counter value
//   NC-Task 1 SAF/Axes/Axis 8(FM-Y3) <-> Device 1 (EtherCAT)/Term 9 (EK1100)/Term 12 (EL2522)
//     Drive/Inputs/In/nState1 @bit 6 <-> PTO Status Channel 1/Status/Error
//     Drive/Inputs/In/nState1 @bit 1 <-> PTO Status Channel 1/Status/Ramp active
//     Drive/Inputs/In/nState1 <-> PTO Status Channel 1/Status/Sel. Ack/End counter
//     Drive/Inputs/In/nState2 @bit 5 <-> PTO Status Channel 1/Status/Sync error
//     Drive/Inputs/In/nState2 @bit 7 <-> PTO Status Channel 1/Status/TxPDO Toggle
//     Drive/Inputs/In/nState4 @bit 1 <-> WcState/InputToggle
//     Drive/Inputs/In/nState4 <-> WcState/WcState
//     Drive/Outputs/Out/nCtrl1 @bit 1 <-> PTO Control Channel 1/Control/Disable ramp
//     Drive/Outputs/Out/nCtrl1 <-> PTO Control Channel 1/Control/Frequency select
//     Drive/Outputs/Out/nCtrl1 @bit 2 <-> PTO Control Channel 1/Control/Go counter
//     Drive/Outputs/Out/nDataOut1[0] <-> PTO Control Channel 1/Frequency value
//     Drive/Outputs/Out/nDataOut5 <-> PTO Target Channel 1/Target counter value
//   NC-Task 1 SAF/Axes/Axis 8(FM-Y3) <-> Device 1 (EtherCAT)/Term 9 (EK1100)/Term 13 (EL5112)
//     Enc/Inputs/In/nDataIn1 <-> ENC Status Channel 1/Counter value
//     Enc/Inputs/In/nDataIn2 <-> ENC Status Channel 1/Latch value
//     Enc/Inputs/In/nState1 @bit 4 <-> ENC Status Channel 1/Status/Counter overflow
//     Enc/Inputs/In/nState1 @bit 3 <-> ENC Status Channel 1/Status/Counter underflow
//     Enc/Inputs/In/nState1 @bit 7 <-> ENC Status Channel 1/Status/Extrapolation stall
//     Enc/Inputs/In/nState1 <-> ENC Status Channel 1/Status/Latch C valid
//     Enc/Inputs/In/nState1 @bit 1 <-> ENC Status Channel 1/Status/Latch extern valid
//     Enc/Inputs/In/nState1 @bit 6 <-> ENC Status Channel 1/Status/Open circuit
//     Enc/Inputs/In/nState1 @bit 2 <-> ENC Status Channel 1/Status/Set counter done
//     Enc/Inputs/In/nState1 @bit 5 <-> ENC Status Channel 1/Status/Status of input status
//     Enc/Inputs/In/nState2 @bit 4 <-> ENC Status Channel 1/Status/Diag
//     Enc/Inputs/In/nState2 @bit 6 <-> ENC Status Channel 1/Status/Input cycle counter
//     Enc/Inputs/In/nState2 <-> ENC Status Channel 1/Status/Status of input A
//     Enc/Inputs/In/nState2 @bit 1 <-> ENC Status Channel 1/Status/Status of input B
//     Enc/Inputs/In/nState2 @bit 2 <-> ENC Status Channel 1/Status/Status of input C
//     Enc/Inputs/In/nState2 @bit 3 <-> ENC Status Channel 1/Status/Status of input gate
//     Enc/Inputs/In/nState2 @bit 5 <-> ENC Status Channel 1/Status/TxPDO State
//     Enc/Inputs/In/nState3 @bit 4 <-> ENC Status Channel 1/Status/Counter value out of range
//     Enc/Inputs/In/nState3 @bit 2 <-> ENC Status Channel 1/Status/Direction inversion detected
//     Enc/Inputs/In/nState3 @bit 1 <-> ENC Status Channel 1/Status/Latch extern 2 valid
//     Enc/Inputs/In/nState3 <-> ENC Status Channel 1/Status/Software gate valid
//     Enc/Inputs/In/nState3 @bit 3 <-> ENC Status Channel 1/Status/Status of extern latch
//     Enc/Inputs/In/nState4 @bit 1 <-> WcState/InputToggle
//     Enc/Inputs/In/nState4 <-> WcState/WcState
//     Enc/Outputs/Out/nCtrl1 <-> ENC Control Channel 1/Control/Enable latch C
//     Enc/Outputs/Out/nCtrl1 @bit 3 <-> ENC Control Channel 1/Control/Enable latch extern on negative edge
//     Enc/Outputs/Out/nCtrl1 @bit 1 <-> ENC Control Channel 1/Control/Enable latch extern on positive edge
//     Enc/Outputs/Out/nCtrl1 @bit 2 <-> ENC Control Channel 1/Control/Set counter
//     Enc/Outputs/Out/nCtrl1 @bit 7 <-> ENC Control Channel 1/Control/Set counter on latch C
//     Enc/Outputs/Out/nCtrl2 @bit 4 <-> ENC Control Channel 1/Control/Enable latch extern 2 on negative edge
//     Enc/Outputs/Out/nCtrl2 @bit 3 <-> ENC Control Channel 1/Control/Enable latch extern 2 on positive edge
//     Enc/Outputs/Out/nCtrl2 @bit 2 <-> ENC Control Channel 1/Control/Set counter on latch extern on negative edge
//     Enc/Outputs/Out/nCtrl2 @bit 1 <-> ENC Control Channel 1/Control/Set counter on latch extern on positive edge
//     Enc/Outputs/Out/nCtrl2 <-> ENC Control Channel 1/Control/Set software gate
//     Enc/Outputs/Out/nDataOut1 <-> ENC Control Channel 1/Set counter value
//   NC-Task 1 SAF/Axes/Axis 9(FM-X1) <-> Device 1 (EtherCAT)/Term 9 (EK1100)/Term 12 (EL2522)
//     Drive/Inputs/In/nState1 @bit 6 <-> PTO Status Channel 2/Status/Error
//     Drive/Inputs/In/nState1 @bit 1 <-> PTO Status Channel 2/Status/Ramp active
//     Drive/Inputs/In/nState1 <-> PTO Status Channel 2/Status/Sel. Ack/End counter
//     Drive/Inputs/In/nState2 @bit 5 <-> PTO Status Channel 2/Status/Sync error
//     Drive/Inputs/In/nState2 @bit 7 <-> PTO Status Channel 2/Status/TxPDO Toggle
//     Drive/Inputs/In/nState4 @bit 1 <-> WcState/InputToggle
//     Drive/Inputs/In/nState4 <-> WcState/WcState
//     Drive/Outputs/Out/nCtrl1 @bit 1 <-> PTO Control Channel 2/Control/Disable ramp
//     Drive/Outputs/Out/nCtrl1 <-> PTO Control Channel 2/Control/Frequency select
//     Drive/Outputs/Out/nCtrl1 @bit 2 <-> PTO Control Channel 2/Control/Go counter
//     Drive/Outputs/Out/nDataOut1[0] <-> PTO Control Channel 2/Frequency value
//     Drive/Outputs/Out/nDataOut5 <-> PTO Target Channel 2/Target counter value
//     Enc/Inputs/In/nDataIn1 <-> ENC Status Channel 2/Counter value
//     Enc/Inputs/In/nState1 @bit 4 <-> ENC Status Channel 2/Status/Counter overflow
//     Enc/Inputs/In/nState1 @bit 3 <-> ENC Status Channel 2/Status/Counter underflow
//     Enc/Inputs/In/nState1 @bit 2 <-> ENC Status Channel 2/Status/Set counter done
//     Enc/Inputs/In/nState2 @bit 5 <-> ENC Status Channel 2/Status/Sync error
//     Enc/Inputs/In/nState2 @bit 6 <-> ENC Status Channel 2/Status/TxPDO State
//     Enc/Inputs/In/nState2 @bit 7 <-> ENC Status Channel 2/Status/TxPDO Toggle
//     Enc/Inputs/In/nState4 @bit 1 <-> WcState/InputToggle
//     Enc/Inputs/In/nState4 <-> WcState/WcState
//     Enc/Outputs/Out/nCtrl1 @bit 2 <-> ENC Control Channel 2/Control/Set counter
//     Enc/Outputs/Out/nCtrl2 @bit 7 <-> ENC Control Channel 2/Control/Reserved
//     Enc/Outputs/Out/nDataOut1 <-> ENC Control Channel 2/Set counter value
//   HFM/HFM Instance <-> Device 1 (EtherCAT)/Term 9 (EK1100)/Term 15 (EL1889)
//     PlcTask Inputs/MAIN.bM{6..10}minusLimit <-> Channel {2..10 step 2}/Input  (5 links)
//     PlcTask Inputs/MAIN.bM{6..10}plusLimit <-> Channel {1..9 step 2}/Input  (5 links)
//   HFM/HFM Instance <-> Device 3 (EtherCAT)/Term 1 (EK1100)/Term 7 (EL1889)
//     PlcTask Inputs/MAIN.bM{1..5}minusLimit <-> Channel {2..10 step 2}/Input  (5 links)
//     PlcTask Inputs/MAIN.bM{1..5}plusLimit <-> Channel {1..9 step 2}/Input  (5 links)
//   HFM/HFM Instance <-> NC-Task 1 SAF/Axes/Axis 1(HFM-Y1)
//     PlcTask Inputs/MAIN.M1.Axis.NcToPlc <-> Outputs/ToPlc
//     PlcTask Outputs/MAIN.M1.Axis.PlcToNc <-> Inputs/FromPlc
//   HFM/HFM Instance <-> NC-Task 1 SAF/Axes/Axis 10(FM-X2)
//     PlcTask Inputs/MAIN.M10.Axis.NcToPlc <-> Outputs/ToPlc
//     PlcTask Outputs/MAIN.M10.Axis.PlcToNc <-> Inputs/FromPlc
//   HFM/HFM Instance <-> NC-Task 1 SAF/Axes/Axis 2(HFM-Y2)
//     PlcTask Inputs/MAIN.M2.Axis.NcToPlc <-> Outputs/ToPlc
//     PlcTask Outputs/MAIN.M2.Axis.PlcToNc <-> Inputs/FromPlc
//   HFM/HFM Instance <-> NC-Task 1 SAF/Axes/Axis 3(HFM-Y3)
//     PlcTask Inputs/MAIN.M3.Axis.NcToPlc <-> Outputs/ToPlc
//     PlcTask Outputs/MAIN.M3.Axis.PlcToNc <-> Inputs/FromPlc
//   HFM/HFM Instance <-> NC-Task 1 SAF/Axes/Axis 4(HFM-X1)
//     PlcTask Inputs/MAIN.M4.Axis.NcToPlc <-> Outputs/ToPlc
//     PlcTask Outputs/MAIN.M4.Axis.PlcToNc <-> Inputs/FromPlc
//   HFM/HFM Instance <-> NC-Task 1 SAF/Axes/Axis 5(HFM-X2)
//     PlcTask Inputs/MAIN.M5.Axis.NcToPlc <-> Outputs/ToPlc
//     PlcTask Outputs/MAIN.M5.Axis.PlcToNc <-> Inputs/FromPlc
//   HFM/HFM Instance <-> NC-Task 1 SAF/Axes/Axis 6(FM-Y1)
//     PlcTask Inputs/MAIN.M6.Axis.NcToPlc <-> Outputs/ToPlc
//     PlcTask Outputs/MAIN.M6.Axis.PlcToNc <-> Inputs/FromPlc
//   HFM/HFM Instance <-> NC-Task 1 SAF/Axes/Axis 7(FM-Y2)
//     PlcTask Inputs/MAIN.M7.Axis.NcToPlc <-> Outputs/ToPlc
//     PlcTask Outputs/MAIN.M7.Axis.PlcToNc <-> Inputs/FromPlc
//   HFM/HFM Instance <-> NC-Task 1 SAF/Axes/Axis 8(FM-Y3)
//     PlcTask Inputs/MAIN.M8.Axis.NcToPlc <-> Outputs/ToPlc
//     PlcTask Outputs/MAIN.M8.Axis.PlcToNc <-> Inputs/FromPlc
//   HFM/HFM Instance <-> NC-Task 1 SAF/Axes/Axis 9(FM-X1)
//     PlcTask Inputs/MAIN.M9.Axis.NcToPlc <-> Outputs/ToPlc
//     PlcTask Outputs/MAIN.M9.Axis.PlcToNc <-> Inputs/FromPlc
//   (this object) <-> Device 3 (EtherCAT)/Term 1 (EK1100)/Term 2 (EL2522)
//     Drive/Inputs/In/nState1 @bit 6 <-> PTO Status Channel 1/Status/Error
//     Drive/Inputs/In/nState1 @bit 1 <-> PTO Status Channel 1/Status/Ramp active
//     Drive/Inputs/In/nState1 <-> PTO Status Channel 1/Status/Sel. Ack/End counter
//     Drive/Inputs/In/nState2 @bit 5 <-> PTO Status Channel 1/Status/Sync error
//     Drive/Inputs/In/nState2 @bit 7 <-> PTO Status Channel 1/Status/TxPDO Toggle
//     Drive/Inputs/In/nState4 @bit 1 <-> WcState/InputToggle
//     Drive/Inputs/In/nState4 <-> WcState/WcState
//     Drive/Outputs/Out/nCtrl1 @bit 1 <-> PTO Control Channel 1/Control/Disable ramp
//     Drive/Outputs/Out/nCtrl1 <-> PTO Control Channel 1/Control/Frequency select
//     Drive/Outputs/Out/nCtrl1 @bit 2 <-> PTO Control Channel 1/Control/Go counter
//     Drive/Outputs/Out/nDataOut1[0] <-> PTO Control Channel 1/Frequency value
//     Drive/Outputs/Out/nDataOut5 <-> PTO Target Channel 1/Target counter value
//   (this object) <-> Device 3 (EtherCAT)/Term 1 (EK1100)/Term 3 (EL5112)
//     Enc/Inputs/In/nDataIn1 <-> ENC Status Channel 1/Counter value
//     Enc/Inputs/In/nDataIn2 <-> ENC Status Channel 1/Latch value
//     Enc/Inputs/In/nState1 @bit 4 <-> ENC Status Channel 1/Status/Counter overflow
//     Enc/Inputs/In/nState1 @bit 3 <-> ENC Status Channel 1/Status/Counter underflow
//     Enc/Inputs/In/nState1 @bit 1 <-> ENC Status Channel 1/Status/Latch extern valid
//     Enc/Inputs/In/nState1 @bit 6 <-> ENC Status Channel 1/Status/Open circuit
//     Enc/Inputs/In/nState1 @bit 2 <-> ENC Status Channel 1/Status/Set counter done
//     Enc/Inputs/In/nState2 @bit 4 <-> ENC Status Channel 1/Status/Diag
//     Enc/Inputs/In/nState2 @bit 6 <-> ENC Status Channel 1/Status/Input cycle counter
//     Enc/Inputs/In/nState2 <-> ENC Status Channel 1/Status/Status of input A
//     Enc/Inputs/In/nState2 @bit 1 <-> ENC Status Channel 1/Status/Status of input B
//     Enc/Inputs/In/nState2 @bit 3 <-> ENC Status Channel 1/Status/Status of input gate
//     Enc/Inputs/In/nState2 @bit 5 <-> ENC Status Channel 1/Status/TxPDO State
//     Enc/Inputs/In/nState3 @bit 4 <-> ENC Status Channel 1/Status/Counter value out of range
//     Enc/Inputs/In/nState3 <-> ENC Status Channel 1/Status/Software gate valid
//     Enc/Inputs/In/nState4 @bit 1 <-> WcState/InputToggle
//     Enc/Inputs/In/nState4 <-> WcState/WcState
//     Enc/Outputs/Out/nCtrl1 @bit 3 <-> ENC Control Channel 1/Control/Enable latch extern on negative edge
//     Enc/Outputs/Out/nCtrl1 @bit 1 <-> ENC Control Channel 1/Control/Enable latch extern on positive edge
//     Enc/Outputs/Out/nCtrl1 @bit 2 <-> ENC Control Channel 1/Control/Set counter
//     Enc/Outputs/Out/nCtrl2 @bit 2 <-> ENC Control Channel 1/Control/Set counter on latch extern on negative edge
//     Enc/Outputs/Out/nCtrl2 @bit 1 <-> ENC Control Channel 1/Control/Set counter on latch extern on positive edge
//     Enc/Outputs/Out/nCtrl2 <-> ENC Control Channel 1/Control/Set software gate
//     Enc/Outputs/Out/nDataOut1 <-> ENC Control Channel 1/Set counter value

CONFIGURATION HFM
    RESOURCE PLC ON TwinCAT3
        TASK PlcTask(INTERVAL := T#10ms, PRIORITY := 20);
        PROGRAM MAIN WITH PlcTask : MAIN;
    END_RESOURCE
END_CONFIGURATION

// ---- POUs/MAIN.TcPOU
PROGRAM MAIN
VAR
	// M1 - HFM Y1
	// M2 - HFM Y2
	// M3 - HFM Y3
	// M4 - HFM X1: RING + / HALL-
	// M5 - HFM X2: RING + / HALL-

	// M6 - FM Y1
	// M7 - FM Y2
	// M8 - FM Y3
	// M9 - FM X1: RING + / HALL-
	// M10 - FM X2: RING + / HALL-	
    
	// M1: ST_MotionStage := (fVelocity:=1.0, nEnableMode:=ENUM_StageEnableMode.DURING_MOTION, bPowerSelf:=TRUE, nHomingMode:=ENUM_EpicsHomeCmd.ABSOLUTE_SET);
	M1: ST_MotionStage := (fVelocity:=1.0, nEnableMode:=ENUM_StageEnableMode.ALWAYS, bPowerSelf:=TRUE, nHomingMode:=ENUM_EpicsHomeCmd.ABSOLUTE_SET);
	fbMotion1: FB_MotionStage;
	bM1plusLimit AT %I*: BOOL;
	bM1minusLimit AT %I*: BOOL;	
	
	M2: ST_MotionStage := (fVelocity:=1.0, nEnableMode:=ENUM_StageEnableMode.ALWAYS, bPowerSelf:=TRUE, nHomingMode:=ENUM_EpicsHomeCmd.ABSOLUTE_SET);
	fbMotion2: FB_MotionStage;
	bM2plusLimit AT %I*: BOOL;
	bM2minusLimit AT %I*: BOOL;	
	
	M3: ST_MotionStage := (fVelocity:=1.0, nEnableMode:=ENUM_StageEnableMode.ALWAYS, bPowerSelf:=TRUE, nHomingMode:=ENUM_EpicsHomeCmd.ABSOLUTE_SET);
	fbMotion3: FB_MotionStage;
	bM3plusLimit AT %I*: BOOL;
	bM3minusLimit AT %I*: BOOL;	
	
	M4: ST_MotionStage := (fVelocity:=1.0, nEnableMode:=ENUM_StageEnableMode.ALWAYS, bPowerSelf:=TRUE, nHomingMode:=ENUM_EpicsHomeCmd.ABSOLUTE_SET);
	fbMotion4: FB_MotionStage;
	bM4plusLimit AT %I*: BOOL;
	bM4minusLimit AT %I*: BOOL;	
	
	M5: ST_MotionStage := (fVelocity:=1.0, nEnableMode:=ENUM_StageEnableMode.ALWAYS, bPowerSelf:=TRUE, nHomingMode:=ENUM_EpicsHomeCmd.ABSOLUTE_SET);
	fbMotion5: FB_MotionStage;
	bM5plusLimit AT %I*: BOOL;
	bM5minusLimit AT %I*: BOOL;	
	
	M6: ST_MotionStage := (fVelocity:=1.0, nEnableMode:=ENUM_StageEnableMode.ALWAYS, bPowerSelf:=TRUE, nHomingMode:=ENUM_EpicsHomeCmd.ABSOLUTE_SET);
	fbMotion6: FB_MotionStage;
	bM6plusLimit AT %I*: BOOL;
	bM6minusLimit AT %I*: BOOL;	
	
	M7: ST_MotionStage := (fVelocity:=1.0, nEnableMode:=ENUM_StageEnableMode.ALWAYS, bPowerSelf:=TRUE, nHomingMode:=ENUM_EpicsHomeCmd.ABSOLUTE_SET);
	fbMotion7: FB_MotionStage;
	bM7plusLimit AT %I*: BOOL;
	bM7minusLimit AT %I*: BOOL;	
	
	M8: ST_MotionStage := (fVelocity:=1.0, nEnableMode:=ENUM_StageEnableMode.ALWAYS, bPowerSelf:=TRUE, nHomingMode:=ENUM_EpicsHomeCmd.ABSOLUTE_SET);
	fbMotion8: FB_MotionStage;
	bM8plusLimit AT %I*: BOOL;
	bM8minusLimit AT %I*: BOOL;	
	
	M9: ST_MotionStage := (fVelocity:=1.0, nEnableMode:=ENUM_StageEnableMode.ALWAYS, bPowerSelf:=TRUE, nHomingMode:=ENUM_EpicsHomeCmd.ABSOLUTE_SET);
	fbMotion9: FB_MotionStage;
	bM9plusLimit AT %I*: BOOL;
	bM9minusLimit AT %I*: BOOL;	
	
	M10: ST_MotionStage := (fVelocity:=1.0, nEnableMode:=ENUM_StageEnableMode.ALWAYS, bPowerSelf:=TRUE, nHomingMode:=ENUM_EpicsHomeCmd.ABSOLUTE_SET);
	fbMotion10: FB_MotionStage;
	bM10plusLimit AT %I*: BOOL;
	bM10minusLimit AT %I*: BOOL;	
	
END_VAR



fbMotion1(stMotionStage := M1);
M1.bError := FALSE;
M1.bHardwareEnable := TRUE;
M1.bPowerSelf := TRUE;
M1.bLimitForwardEnable := bM1plusLimit;
M1.bLimitBackwardEnable := bM1minusLimit;

fbMotion2(stMotionStage := M2);
M2.bError := FALSE;
M2.bHardwareEnable := TRUE;
M2.bPowerSelf := TRUE;
M2.bLimitForwardEnable := bM2plusLimit;
M2.bLimitBackwardEnable := bM2minusLimit;

fbMotion3(stMotionStage := M3);
M3.bError := FALSE;
M3.bHardwareEnable := TRUE;
M3.bPowerSelf := TRUE;
M3.bLimitForwardEnable := bM3plusLimit;
M3.bLimitBackwardEnable := bM3minusLimit;

fbMotion4(stMotionStage := M4);
M4.bError := FALSE;
M4.bHardwareEnable := TRUE;
M4.bPowerSelf := TRUE;
M4.bLimitForwardEnable := bM4plusLimit;
M4.bLimitBackwardEnable := bM4minusLimit;

fbMotion5(stMotionStage := M5);
M5.bError := FALSE;
M5.bHardwareEnable := TRUE;
M5.bPowerSelf := TRUE;
M5.bLimitForwardEnable := bM5plusLimit;
M5.bLimitBackwardEnable := bM5minusLimit;

fbMotion6(stMotionStage := M6);
M6.bError := FALSE;
M6.bHardwareEnable := TRUE;
M6.bPowerSelf := TRUE;
M6.bLimitForwardEnable := bM6plusLimit;
M6.bLimitBackwardEnable := bM6minusLimit;

fbMotion7(stMotionStage := M7);
M7.bError := FALSE;
M7.bHardwareEnable := TRUE;
M7.bPowerSelf := TRUE;
M7.bLimitForwardEnable := bM7plusLimit;
M7.bLimitBackwardEnable := bM7minusLimit;

fbMotion8(stMotionStage := M8);
M8.bError := FALSE;
M8.bHardwareEnable := TRUE;
M8.bPowerSelf := TRUE;
M8.bLimitForwardEnable := bM8plusLimit;
M8.bLimitBackwardEnable := bM8minusLimit;

fbMotion9(stMotionStage := M9);
M9.bError := FALSE;
M9.bHardwareEnable := TRUE;
M9.bPowerSelf := TRUE;
M9.bLimitForwardEnable := bM9plusLimit;
M9.bLimitBackwardEnable := bM9minusLimit;

fbMotion10(stMotionStage := M10);
M10.bError := FALSE;
M10.bHardwareEnable := TRUE;
M10.bPowerSelf := TRUE;
M10.bLimitForwardEnable := bM10plusLimit;
M10.bLimitBackwardEnable := bM10minusLimit;

END_PROGRAM
